(* IEC 61131-3 sources: inproshop/test9_exported/OP60/1.Global, 6 files *)

(* ---- DB6000_Control.st ---- *)
VAR_GLOBAL
	Mode:Str_Mode;
	HMI:Str_HMI;
END_VAR
VAR_GLOBAL RETAIN PERSISTENT
	Machine AT %MB132436 : Str_Machine;
END_VAR

(* ---- DB6003_Count.st ---- *)
VAR_GLOBAL RETAIN PERSISTENT
	Total AT %MB178016 : Str_Count;//总计数
	OK AT %MB178688 : Str_Count;//OK计数
	NG AT %MB235528 : Str_Count;//NG计数
END_VAR
VAR_GLOBAL
	Yield : REAL;//良品率
	Clear : BOOL;//清除计数
END_VAR

(* ---- DB6005_Communication.st ---- *)
VAR_GLOBAL
	TcpClient:ARRAY[0..9] OF Str_TcpClient;
	TcpSever:ARRAY[0..9] OF Str_TcpClient;
	From_OPXX    :Str_OP80_TO_OPXX;
	TO_OPXX    :Str_OPXX_TO_OP80;
	FromMaster  :Str_FromMaster;
END_VAR

(* ---- DB6050_DriveControl.st ---- *)
VAR_GLOBAL RETAIN PERSISTENT
	CylCtrl AT %MB329164 : ARRAY [0..63] OF Str_Cylinder;
	VacCtrl AT %MB399516 : ARRAY [0..32] OF Str_Cylinder;
	AxisCtrl AT %MB403940 : ARRAY [0..16] OF Str_Axis;
	Sensor AT %MB433180 : ARRAY [0..32] OF Str_Sensor;
	CamCtrl AT %MB146692 : ARRAY [1..3] OF Str_CamControl;
END_VAR

VAR_GLOBAL
	DoubleStart:ARRAY [1..4] OF Str_DoubleStart;
	Epson : ARRAY [1..10] OF Str_Epson;
	Kuka : ARRAY [1..2] OF Str_Kuka6;
	Rotdisk:ARRAY [1..1] OF Str_Rotdisk;
	Stopper:ARRAY [1..20] OF Str_Stopper;
	Motor:ARRAY [1..10] OF Str_Motor;
	AI:ARRAY [0..20] OF Str_AI;
	AAS:ARRAY [1..1] OF Str_AAS;
	HeatCtrl : ARRAY [1..1] OF Str_Heating;
	PalletCtrl : ARRAY [0..3] OF Str_Palletizing;
END_VAR

(* ---- DB6070_Fault.st ---- *)
VAR_GLOBAL
	Estop:Str_OP30_FaultEstop;//紧急停止类报警
	Stop:Str_OP30_Faultstop;//暂停类报警
	Run:Str_OP30_FaultRun;//警告类报警
	EstopTotal:BOOL;//急停报警汇总
	StopTotal:BOOL;//暂停报警汇总
	RunTotal:BOOL;//警告汇总
END_VAR

(* ---- DB6090_Other.st ---- *)
VAR_GLOBAL RETAIN PERSISTENT
	{attribute 'ElemComment':='(),(上料机械臂取料夹爪),(上料机械臂放料夹爪),(缓存台1),(缓存台2),(缓存台3),(缓存台4),(测试台1),(测试台2),(测试台3),(测试台4),(下料机械臂),4()'}
	StationData AT %MB326468 : ARRAY [0..15] OF Str_OP30_StationData;
END_VAR
